Staubli VAL3: onF8Event.pgx

program onF8Event()
  local string l_sNew
  local bool l_bUndo
  local num l_nResult
begin
//  // look if the bButton is enable
  if bButton[7]
    call cycle:wizard()
    call buildList()
  endIf
end
